// TIA Portal V20 export
TYPE "LER_typeStatusEm3"
// stored: Access Published
   STRUCT
      compensatorCamEnabled : Bool;
      unwinderGearEnabled : Bool;
      stackJobCompleteChecked : Bool;
      calculateDiameter : Bool;
      sequenceComplete : Bool;
      stopRequest : Bool;
      stopStart : Bool;
      stopComplete : Bool;
      compensatorOffset : LReal;
      compensatorStart : LReal := 0.0;
      compensatorEnd : LReal := 75.0;
      compensatorStartOffset : LReal;
      preCount : LReal;
      prePosition : LReal;
      targetPosition : LReal;
      PretargetPosition : LReal;
      PreReelCutTargetCount : LReal;
      UnwinderGearRatio : DInt := 10000;
      unwinderDelay : Time;
      CompansatorAutoReadyDis : LReal;
   END_STRUCT;
END_TYPE
